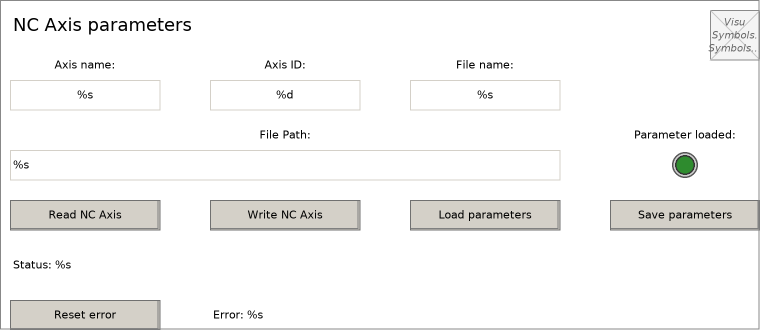
VISUALIZATION NcParameterHandler_View  // 760x330
VAR_IN_OUT
	DataContent: NcParameterHandler_ViewModel;
END_VAR
    Button (10,200 150x30), "Read NC Axis", tooltip "Read the parameters from the NC Axis"
        tap DataContent.ReadButton
    Textfield (10,80 150x30), "%s", tooltip "Axis name to be saved in the JSON file.", text variable: DataContent.AxisName
        OnMouseClick: write the text variable via Default
    Label (10,50 150x30), "Axis name:"
    Button (210,200 150x30), "Write NC Axis", tooltip "Write the parameters to the NC Axis"
        tap DataContent.WriteButton
    Button (410,200 150x30), "Load parameters", tooltip "Load the parameters from the JSON file"
        tap DataContent.LoadButton
    Button (610,200 150x30), "Save parameters", tooltip "Save the parameters to the JSON file"
        tap DataContent.SaveButton
    Label (210,50 150x30), "Axis ID:"
    Textfield (210,80 150x30), "%d", tooltip "The axis ID in the Motion controller under the General tab.", text variable: DataContent.AxisId
        OnMouseClick: write the text variable via Default
    Label (10,120 550x30), "File Path:"
    Textfield (10,150 550x30), "%s", tooltip "Path to where the JSON parameter file is loaded from and saved to.", text variable: DataContent.ParameterPath
        OnMouseClick: write the text variable via Default
    Label (10,10 350x30), "NC Axis parameters"
    Textfield (10,250 200x30), "Status: %s", text variable: DataContent.Status
    Textfield (210,300 550x30), "Error: %s", text variable: DataContent.ErrorString, invisible if: NOT DataContent.Error
    Button (10,300 150x30), "Reset error", tooltip "Reset any error that occured", invisible if: NOT DataContent.Error
        tap DataContent.ResetButton
    Label (410,50 150x30), "File name:"
    Textfield (410,80 150x30), "%s", tooltip "File name for the JSON to be saved to. White space it not allowed in the name. .json file extension is concated on the name.", text variable: DataContent.FileName
        OnMouseClick: write the text variable via Default
    Image (710,10 50x50), tooltip "This Visu can be used for reading and writing to the NC Axis in the Motion controller. It can also load and save the parameter to a JSON file on the OS. To read and write the NC parameter, you need to provide a AxisID. To load and save the parameter, you need to provide the file name and path to the file.", image: VisuSymbols.Symbols.Information
    Lamp1 (670,150 30x30), tooltip "Indicate if a parameter set have been loaded or read into the Visu.", variable: DataContent.ParameterLoaded, style: Lamp-Lamp1-Green
    Label (610,120 150x30), "Parameter loaded:"
END_VISUALIZATION

(* stored: Version 1.1.0.1, ProductVersion 3.1.4026.18
   Visu NcParameterHandler_View: Id {076a4b2a-0e64-0767-1e52-6e167d8958e4} *)
